FUNCTION_BLOCK DS_SELECTX_2536758B411A6CE51 (* Service Interface Function Block Type *)
  (* Standard: 61499-2 *)
  (* Version 1.0, 06.02.2012, hoegdan, nxtControl GmbH, Initial Version *)
  PACKAGE UAO.Hackathon;
  (* Compiler Cpp nxtControl builtin 1.0 *)
  {SET_ATTRIBUTE(Runtime.FBType.ImplementingType, Runtime.Standard#DYNGEN_DS_SELECT)}
  {SET_ATTRIBUTE(Configuration.GenericFBType.InterfaceParams, Runtime.Standard#CNTX:=2;CNTY:=1;DI${CNTX,_,CNTY$}:BOOL)}
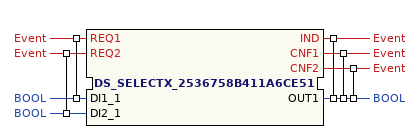
  EVENT_INPUT
    REQ1 WITH DI1_1; (* Request events for dedicated input data sets *)
    REQ2 WITH DI2_1; (* Request events for dedicated input data sets *)
  END_EVENT
  EVENT_OUTPUT
    IND WITH OUT1; (* Indication from Resource *)
    CNF1 WITH OUT1; (* Confirmation from Resource for a dedicated request *)
    CNF2 WITH OUT1; (* Confirmation from Resource for a dedicated request *)
  END_EVENT
  VAR_INPUT
    DI1_1 : BOOL; (* Output data to resource *)
    DI2_1 : BOOL; (* Output data to resource *)
  END_VAR
  VAR_OUTPUT
    OUT1 : BOOL; (* Input data from resource *)
  END_VAR
  EC_STATES
    START;
  END_STATES
END_FUNCTION_BLOCK
